FUNCTION_BLOCK FB_Test
VAR
	nCounters : LINT;
END_VAR

nCounter := nCounter + 1;

END_FUNCTION_BLOCK

(* stored: Version 1.1.0.1, ProductVersion 3.1.4024.12
   POU FB_Test: Id {c45e2ec8-cfb3-4a34-b853-db771b582e5e}, SpecialFunc None *)
